TYPE (* A service query form for the Arrowhead framework 4.0 *)
  (* Standard: 61499-2; Description: Copyright (c) 2019 fortiss GmbH This program and the accompanying materials are made available under the terms of the Eclipse Public License 2.0 which is available at https://www.eclipse.org/legal/epl-2.0/ SPDX-License-Identifier: EPL-2.0 *)
  (* Version 1.0, 2018-09-26, Jose Cabral, fortiss GmbH *)
  (* ASN.1 tag APPLICATION 1 *)
  ServiceQueryForm : STRUCT
    service : ArrowheadService; (* The Arrowhead Service object that is looked for (SD and supported IDD-s) *)
    metadataSearch : BOOL; (* True, if service metadata shall be taken into account during query. *)
    pingProviders : BOOL; (* True, if the selected (query fitting) Application Systems shall be pinged to see if they are alive. *)
    version : DINT; (* The minimum version of the Service we are looking for. *)
  END_STRUCT;
END_TYPE
